ABB RAPID module: pers_calib_vars.mod

MODULE pers_calib_vars
    CONST num calib_array_size := 40;
    PERS robtarget calib_robtargets{calib_array_size};
ENDMODULE
